(* IEC 61131-3 sources: uPC2_EMCTEST/UPC2_EMCTEST/UPC2_EMCTEST/Gui/Actions, 20 files *)

(* ---- CheckPassword.st ---- *)
USING System;
USING System.UI;

VAR_GLOBAL
    (**Saves current time*)
    {ATTRIBUTE UOM MILLISECOND}
    MemTimePwdWrg           : UDINT;
END_VAR

FUNCTION CheckPassword
	VAR_INPUT
		keyPressed:UINT;
		keyCounter:UINT;
	END_VAR
	VAR_IN_OUT
		value:UINT;
	END_VAR

    (* Saves the last digit. *)
    pGD1.GoToNextField();

    WrngPwd := FALSE;
    (* Concatenate the digits to reconstruct the password. *)
    TmpPwd := TmpPwd_Dig1*1000 + TmpPwd_Dig2*100 + TmpPwd_Dig3*10 + TmpPwd_Dig4;

    IF TmpPwd = PwdSys THEN
        Access_Sys      := TRUE;
        LoginPwdType    := LOGIN_PASSWORD#System;
    ELSIF TmpPwd = PwdUser THEN
        Access_User     := TRUE;
        LoginPwdType    := LOGIN_PASSWORD#User;
    ELSIF TmpPwd = PwdService THEN
        Access_Service  := TRUE;
        LoginPwdType    := LOGIN_PASSWORD#Service;
    ELSIF TmpPwd = PwdManuf THEN
        Access_Manuf    := TRUE;
        LoginPwdType    := LOGIN_PASSWORD#Manufacturer;
    ELSE
        WrngPwd         := TRUE;
        MemTimePwdWrg   := CurrSysT;
    END_IF;

    IF Access_User OR Access_Service OR Access_Sys OR Access_Manuf THEN
        pGD1.GoToLoop(pGD1_LoopList#Menu);
    ELSE
        (* Reset. *)
        TmpPwd_Dig1 := 0;
        TmpPwd_Dig2 := 0;
        TmpPwd_Dig3 := 0;
        TmpPwd_Dig4 := 0;

        TmpPwd  := 0;

        (* Repositions the cursor to the first digit. *)
        pGD1.GoToNextField();
    END_IF;

END_FUNCTION

(* ---- Act_GotoMainMSK.st ---- *)
USING System;
USING System.UI;

FUNCTION Act_GotoMainMSK
	VAR_INPUT
		keyPressed:UINT;
		keyCounter:UINT;
	END_VAR

    pGD1.GoToMask(pGD1_MaskList#MainMask);
END_FUNCTION

(* ---- AskPwd.st ---- *)
USING System;
USING System.UI;

(**Ask password when pressed PRG key*)
FUNCTION AskPwd
	VAR_INPUT
		keyPressed:UINT;
		keyCounter:UINT;
	END_VAR

    {REGION CHECK IF USER IS LOGGED}
        Req_FixLED_PRG := TRUE;

        // Reset
        TmpPwd_Dig1 := 0;
        TmpPwd_Dig2 := 0;
        TmpPwd_Dig3 := 0;
        TmpPwd_Dig4 := 0;

        TmpPwd  := 0;

       // pGD1.MenuWidget.ResetWidget();
        MenuWidget1.ResetWidget();

        (*Check LogIn password, and if necessary asks to insert password*)
        IF Access_User OR Access_Service OR Access_Manuf OR Access_Sys THEN
            pGD1.GoToLoop(pGD1_LoopList#Menu);
        ELSE
            WrngPwd := FALSE;
            pGD1.GoToLoop(pGD1_LoopList#Login);
        END_IF;
    {ENDREGION}

END_FUNCTION

(* ---- ChangeDateFormatENTER.st ---- *)
USING System;
USING System.UI;

FUNCTION ChangeDateFormatENTER
	VAR_INPUT
		keyPressed:UINT;
		keyCounter:UINT;
	END_VAR
	VAR_IN_OUT
		value:USINT;
	END_VAR

    VAR
        MyDateFrmt : DateFormat;
    END_VAR

    MyDateFrmt := TO_USINT(value);

    GetDate_From_DateFormat(MyDateFrmt, LocDateAndTime, DateTimeBypGD1.Hour, DateTimeBypGD1.Minute, DateTimeBypGD1.Second, DateP1, DateP1Lmin, DateP1Lmax, DateP2, DateP2Lmin, DateP2Lmax, DateP3, DateP3Lmin, DateP3Lmax);

    pGD1.GoToNextField();

END_FUNCTION

(* ---- DoNothing.st ---- *)
USING System;
USING System.UI;

FUNCTION DoNothing
	VAR_INPUT
		keyPressed:UINT;
		keyCounter:UINT;
	END_VAR

END_FUNCTION

(* ---- GoToLoopAlarms.st ---- *)
USING System;
USING System.UI;

FUNCTION GoToLoopAlarms
	VAR_INPUT
		keyPressed:UINT;
		keyCounter:UINT;
	END_VAR

//    IF NOT EnLangMskCdwnT THEN                          (*At the 1st SW start up the LANGUAGE Mask has Key-ALARM disabled. *)

        {REGION Buzzer and Led Alarm}
            BuzzerSilenced     := TRUE;
            (*Stop blink of LED alarm*)
            Req_BlinkLED_Alarm := FALSE;
            (*Stop blink of LED alarm*)
            Req_FixLED_Alarm   := GblAlarm;

            Req_FixLED_PRG := FALSE;
        {ENDREGION}

        {REGION Reset Menu and SubMenu}
            MenuWidget1.ResetWidget();
            SubMenuWidget1.ResetWidget();
        {ENDREGION}

        pGD1.GoToLoop(pGD1_LoopList#Alarms);
//    END_IF;
END_FUNCTION

(* ---- GoToMainLoop.st ---- *)
USING System;
USING System.UI;

FUNCTION GoToMainLoop
	VAR_INPUT
		keyPressed:UINT;
		keyCounter:UINT;
	END_VAR

    Req_FixLED_PRG := FALSE;
    pGD1.GoToLoop(pGD1_LoopList#Main);
END_FUNCTION

(* ---- GoToPreviousDigit.st ---- *)
USING System;
USING System.UI;

FUNCTION GoToPreviousDigit
	VAR_INPUT
		keyPressed:UINT;
		keyCounter:UINT;
	END_VAR

    VAR
        i : INT;
    END_VAR

    FOR i := 1 TO 4 DO
        pGD1.GoToNextField();
    END_FOR;
END_FUNCTION

(* ---- LogOutMskENTER.st ---- *)
USING System;
USING System.UI;

FUNCTION LogOutMskENTER
	VAR_INPUT
		keyPressed:UINT;
		keyCounter:UINT;
	END_VAR

    {REGION RESET ACCESS}
        Access_Sys      := FALSE;
        Access_User     := FALSE;
        Access_Service := FALSE;
        Access_Manuf    := FALSE;
    {ENDREGION}

    MenuWidget1.ResetWidget();
    pGD1.GoToLoop(pGD1_LoopList#Main);
END_FUNCTION

(* ---- MainMenuALARM.st ---- *)
USING System;
USING System.UI;

FUNCTION MainMenuALARM
	VAR_INPUT
		keyPressed:UINT;
		keyCounter:UINT;
	END_VAR

    pGD1.GoToLoop(pGD1_LoopList#Language);
END_FUNCTION

(* ---- MainMenuENTER.st ---- *)
USING System;
USING System.UI;

FUNCTION MainMenuENTER
	VAR_INPUT
		keyPressed:UINT;
		keyCounter:UINT;
	END_VAR

    pgd1.GoToLoop(pGD1_LoopList#DateTime);
END_FUNCTION

(* ---- QuickMenuDOWN.st ---- *)
USING System;
USING System.UI;

(** Function for DOWN key of main mask. *)
FUNCTION QuickMenuDOWN
	VAR_INPUT
		keyPressed:UINT;
		keyCounter:UINT;
	END_VAR

    IF IdxQM = QUICK_MENU#OnOff THEN
        IdxQM := QUICK_MENU#Info;
    ELSE
        IdxQM := IdxQM - 1;
    END_IF;
END_FUNCTION

(* ---- QuickMenuENTER.st ---- *)
USING System;
USING System.UI;

(** #Alla pressione del tasto enter accede al loop indicato dal quick menu. *)
FUNCTION QuickMenuENTER
	VAR_INPUT
		keyPressed:UINT;
		keyCounter:UINT;
	END_VAR

    CASE IdxQM OF
        QUICK_MENU#OnOff:
            pGD1.GotoLoop(pGd1_LoopList#ONOFF);

        QUICK_MENU#Set:
            pGD1.GotoLoop(pGd1_LoopList#SET);

        QUICK_MENU#Info:
            pGD1.GotoLoop(pGd1_LoopList#Loop0);
    END_CASE;
END_FUNCTION

(* ---- QuickMenuUP.st ---- *)
USING System;
USING System.UI;

(** Function for UP key of main mask. *)
FUNCTION QuickMenuUP
	VAR_INPUT
		keyPressed:UINT;
		keyCounter:UINT;
	END_VAR

    IF IdxQM = QUICK_MENU#Info THEN
        IdxQM := QUICK_MENU#OnOff;
    ELSE
        IdxQM := IdxQM + 1;
    END_IF;
END_FUNCTION

(* ---- RestoreDefaultENTER.st ---- *)
USING System;
USING System.UI;

FUNCTION RestoreDefaultENTER
	VAR_INPUT
		keyPressed:UINT;
		keyCounter:UINT;
	END_VAR
	VAR_IN_OUT
		value:BOOL;
	END_VAR

    pGD1.GoToNextField();
    IF value THEN
        pGD1.GoToLoop(pGD1_LoopList#DefaultDone);
    END_IF;

END_FUNCTION

(* ---- ReturnToSubMenuSettings.st ---- *)
USING System;
USING System.UI;

FUNCTION ReturnToSubMenuSettings
	VAR_INPUT
		keyPressed:UINT;
		keyCounter:UINT;
	END_VAR
    pGD1.GoToLoop(pGD1_LoopList#SubMenuSettings);

END_FUNCTION

(* ---- ReutrnToMenu.st ---- *)
USING System;
USING System.UI;

FUNCTION ReutrnToMenu
	VAR_INPUT
		keyPressed:UINT;
		keyCounter:UINT;
	END_VAR

    pGD1.GoToLoop(pGD1_LoopList#Menu);
END_FUNCTION

(* ---- SetDateENTER.st ---- *)
USING System;
USING System.UI;

FUNCTION SetDateENTER
	VAR_INPUT
		keyPressed:UINT;
		keyCounter:UINT;
	END_VAR
    VAR_IN_OUT
		value:UINT;
	END_VAR

    SetDate_From_DateFormat(DateFrmt, DateTimeBypGD1.Hour, DateTimeBypGD1.Minute, DateTimeBypGD1.Second, DateP1, DateP2, DateP3);

    pGD1.GoToNextField();
END_FUNCTION

(* ---- UnitOnOffDOWN.st ---- *)
USING System;
USING System.UI;

FUNCTION UnitOnOffDOWN
	VAR_INPUT
		keyPressed:UINT;
		keyCounter:UINT;
	END_VAR

    KeybOnOff := FALSE;
END_FUNCTION

(* ---- UnitOnOffUP.st ---- *)
USING System;
USING System.UI;

FUNCTION UnitOnOffUP
	VAR_INPUT
		keyPressed:UINT;
		keyCounter:UINT;
	END_VAR

    KeybOnOff := TRUE;
END_FUNCTION
